FUNCTION_BLOCK FB_Alarm
VAR_INPUT
	
	//Error/Warning from devices
	safetyRelay : BOOL;
	sensorTimeout : BOOL;
	actuatorWarning : BOOL;
	controllerWarning : BOOL;
	
END_VAR

VAR_OUTPUT
	//Enable system when no error and disable system when error
	sysEnable : BOOL;
	sysHome : BOOL;
	
END_VAR

VAR
	//Operation status to devices
	stopCase : BOOL;
	resetCase : BOOL;
	runCase : BOOL;
	homing : BOOL;
	
END_VAR

//When safety relay active -> stop system and reset system when back to run status.
IF safetyRelay THEN
	stopCase := TRUE;
	sysEnable := FALSE;
	homing := TRUE;
ELSIF homing AND NOT safetyRelay THEN
	sysHome := TRUE;
	resetCase := TRUE;
	sysEnable := TRUE;
	homing := FALSE;
ELSIF NOT safetyRelay AND NOT homing THEN
	sysHome := FALSE;
END_IF

//When sensor timeout -> stop system and continue to run when back to run status.
IF sensorTimeout OR actuatorWarning OR controllerWarning THEN
	sysEnable := FALSE;
	stopCase := TRUE;
ELSE sysEnable := TRUE; runCase := TRUE;
END_IF

// Truong Test Folk

METHOD cylinders : BOOL
VAR_INPUT
END_VAR
END_METHOD

METHOD detectSensors : BOOL
VAR_INPUT
END_VAR
END_METHOD

METHOD doorInterlock : BOOL
VAR_INPUT
END_VAR
END_METHOD

METHOD safetyRelay : BOOL
VAR_INPUT
END_VAR
END_METHOD

METHOD slider : BOOL
VAR_INPUT
END_VAR
END_METHOD

END_FUNCTION_BLOCK

(* stored: Version 1.1.0.1, ProductVersion 3.1.4024.13
   POU FB_Alarm: Id {783ca431-c2ae-4a1a-b212-5b740a356f66}, SpecialFunc None
   Method cylinders: Id {873f6f2d-74fc-4261-a5bc-9c8f56fb6bbc}
   Method detectSensors: Id {5b8ca9e6-36bc-4628-83bb-cda62996a70c}
   Method doorInterlock: Id {b2fe8759-b8a5-4536-843e-2e9a4e6f9227}
   Method safetyRelay: Id {80c48fdf-cfc9-40b0-b1b5-913f6976a038}
   Method slider: Id {396c523d-3740-4243-ab9c-2ec9866fc747} *)
